// LS Electric XG5000 project: LoadWizardPro
// PLC LoadWizardPLC
// module base 0 slot 0: Input Module:XGI-D22A/B (DC 24V Input, 16 Contacts)
// module base 0 slot 1: Output Module:XGQ-RY2A/B (Relay Output, 16 Contacts (2A, No Varistor/Varistor))
// module base 0 slot 2: FEnet:XGL-EFMT(B) (Fast Ethernet Module, Electrical Master)
// module base 0 slot 0: Input/Output Module:XBE-DR16A (DC 24V Input, Relay Output, 16 Contacts)
// module base 0 slot 1: Input/Output Module:XBE-DR16A (DC 24V Input, Relay Output, 16 Contacts)

PROGRAM Main (task: Scan Program)

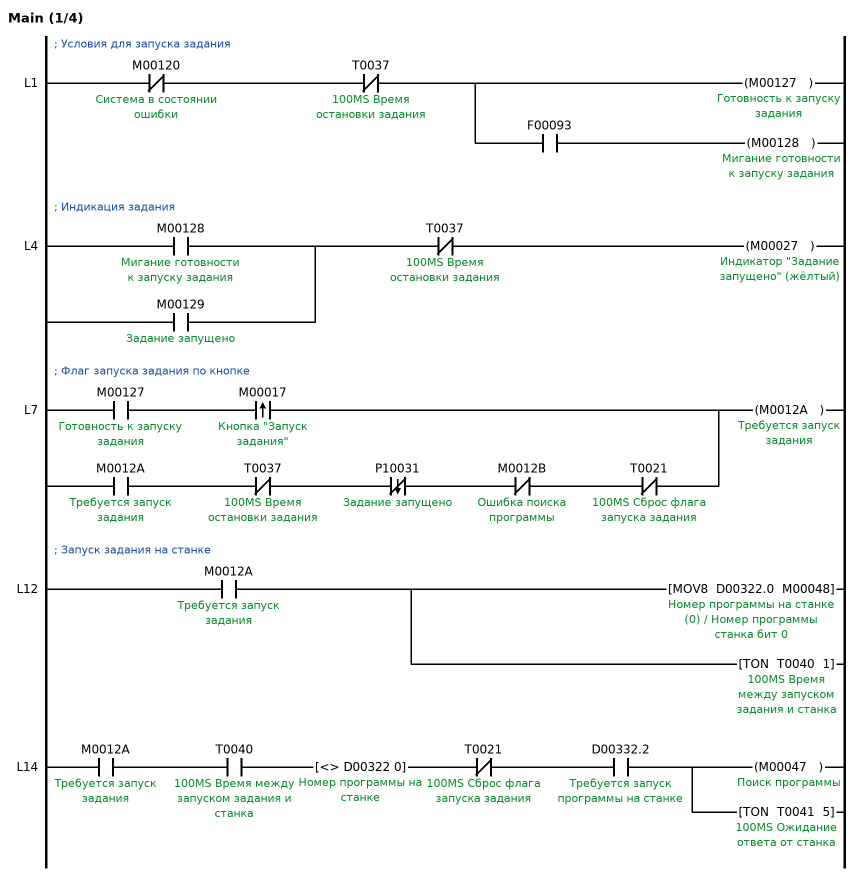
// Условия для запуска задания
; L1
LOAD NOT  M00120	// Система в состоянии ошибки
AND NOT   T0037	// 100MS Время остановки задания
OUT       M00127	// Готовность к запуску задания
AND       F00093
OUT       M00128	// Мигание готовности к запуску задания
// Индикация задания
; L4
LOAD      M00128	// Мигание готовности к запуску задания
OR        M00129	// Задание запущено
AND NOT   T0037	// 100MS Время остановки задания
OUT       M00027	// Индикатор "Задание запущено" (жёлтый)
// Флаг запуска задания по кнопке
; L7
LOAD      M00127	// Готовность к запуску задания
ANDP      M00017	// Кнопка "Запуск задания"
LOAD      M0012A	// Требуется запуск задания
AND NOT   T0037	// 100MS Время остановки задания
ANDN NOT  P10031	// Задание запущено
AND NOT   M0012B	// Ошибка поиска программы
AND NOT   T0021	// 100MS Сброс флага запуска задания
OR LOAD
OUT       M0012A	// Требуется запуск задания
// Запуск задания на станке
; L12
LOAD      M0012A	// Требуется запуск задания
MOV8      D00322.0 M00048	// Номер программы на станке (0) / Номер программы станка бит 0
TON       T0040 1	// 100MS Время между запуском задания и станка
; L14
LOAD      M0012A	// Требуется запуск задания
AND       T0040	// 100MS Время между запуском задания и станка
AND<>     D00322 0	// Номер программы на станке
AND NOT   T0021	// 100MS Сброс флага запуска задания
AND       D00332.2	// Требуется запуск программы на станке
OUT       M00047	// Поиск программы
TON       T0041 5	// 100MS Ожидание ответа от станка

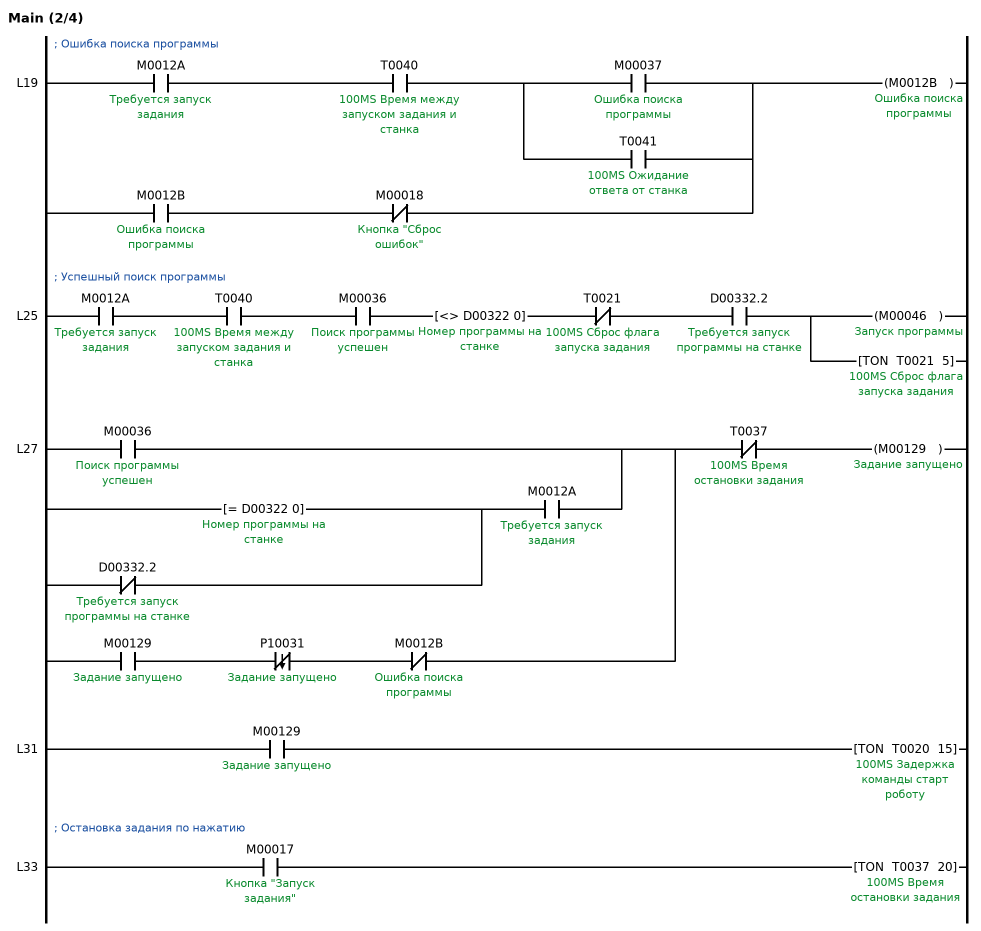
// Ошибка поиска программы
; L19
LOAD      M0012A	// Требуется запуск задания
AND       T0040	// 100MS Время между запуском задания и станка
LOAD      M00037	// Ошибка поиска программы
OR        T0041	// 100MS Ожидание ответа от станка
AND LOAD
LOAD      M0012B	// Ошибка поиска программы
AND NOT   M00018	// Кнопка "Сброс ошибок"
OR LOAD
OUT       M0012B	// Ошибка поиска программы
// Успешный поиск программы
; L25
LOAD      M0012A	// Требуется запуск задания
AND       T0040	// 100MS Время между запуском задания и станка
AND       M00036	// Поиск программы успешен
AND<>     D00322 0	// Номер программы на станке
AND NOT   T0021	// 100MS Сброс флага запуска задания
AND       D00332.2	// Требуется запуск программы на станке
OUT       M00046	// Запуск программы
TON       T0021 5	// 100MS Сброс флага запуска задания
; L27
LOAD      M00036	// Поиск программы успешен
LOAD=     D00322 0	// Номер программы на станке
OR NOT    D00332.2	// Требуется запуск программы на станке
AND       M0012A	// Требуется запуск задания
OR LOAD
LOAD      M00129	// Задание запущено
ANDN NOT  P10031	// Задание запущено
AND NOT   M0012B	// Ошибка поиска программы
OR LOAD
AND NOT   T0037	// 100MS Время остановки задания
OUT       M00129	// Задание запущено
; L31
LOAD      M00129	// Задание запущено
TON       T0020 15	// 100MS Задержка команды старт роботу
// Остановка задания по нажатию
; L33
LOAD      M00017	// Кнопка "Запуск задания"
TON       T0037 20	// 100MS Время остановки задания

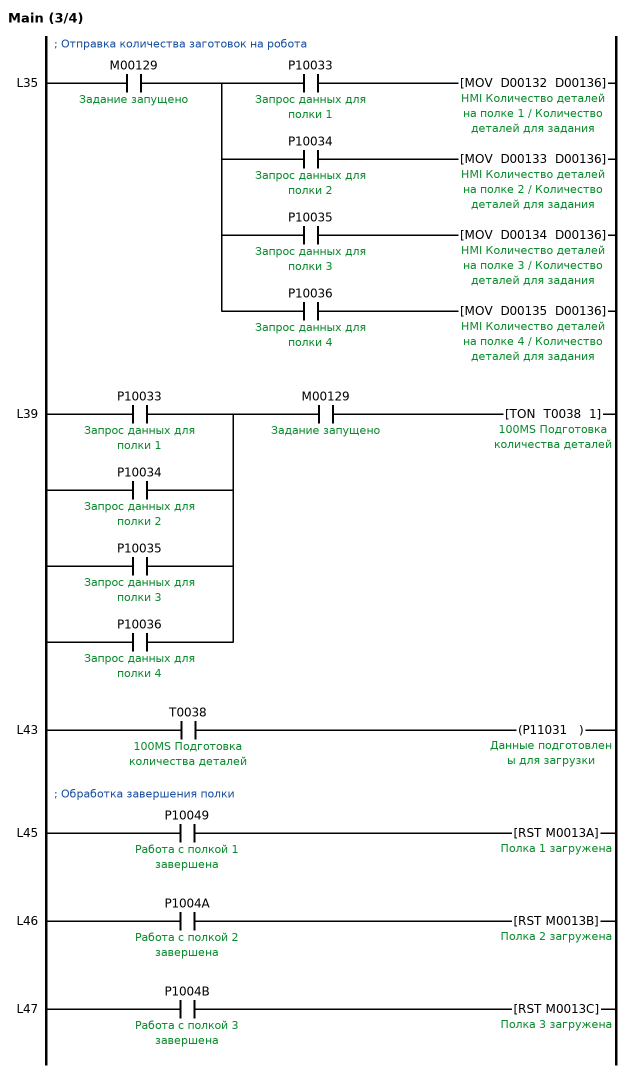
// Отправка количества заготовок на робота
; L35
LOAD      M00129	// Задание запущено
MPUSH
AND       P10033	// Запрос данных для полки 1
MOV       D00132 D00136	// HMI Количество деталей на полке 1 / Количество деталей для задания
MLOAD
AND       P10034	// Запрос данных для полки 2
MOV       D00133 D00136	// HMI Количество деталей на полке 2 / Количество деталей для задания
MLOAD
AND       P10035	// Запрос данных для полки 3
MOV       D00134 D00136	// HMI Количество деталей на полке 3 / Количество деталей для задания
MPOP
AND       P10036	// Запрос данных для полки 4
MOV       D00135 D00136	// HMI Количество деталей на полке 4 / Количество деталей для задания
; L39
LOAD      P10033	// Запрос данных для полки 1
OR        P10034	// Запрос данных для полки 2
OR        P10035	// Запрос данных для полки 3
OR        P10036	// Запрос данных для полки 4
AND       M00129	// Задание запущено
TON       T0038 1	// 100MS Подготовка количества деталей
; L43
LOAD      T0038	// 100MS Подготовка количества деталей
OUT       P11031	// Данные подготовлены для загрузки
// Обработка завершения полки
; L45
LOAD      P10049	// Работа с полкой 1 завершена
RST       M0013A	// Полка 1 загружена
; L46
LOAD      P1004A	// Работа с полкой 2 завершена
RST       M0013B	// Полка 2 загружена
; L47
LOAD      P1004B	// Работа с полкой 3 завершена
RST       M0013C	// Полка 3 загружена

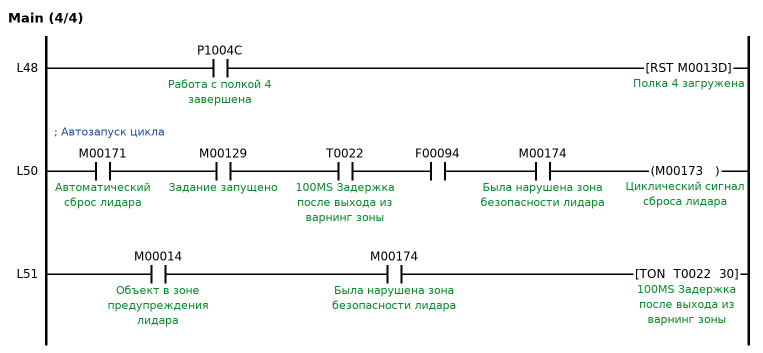
; L48
LOAD      P1004C	// Работа с полкой 4 завершена
RST       M0013D	// Полка 4 загружена
// Автозапуск цикла
; L50
LOAD      M00171	// Автоматический сброс лидара
AND       M00129	// Задание запущено
AND       T0022	// 100MS Задержка после выхода из варнинг зоны
AND       F00094
AND       M00174	// Была нарушена зона безопасности лидара
OUT       M00173	// Циклический сигнал сброса лидара
; L51
LOAD      M00014	// Объект в зоне предупреждения лидара
AND       M00174	// Была нарушена зона безопасности лидара
TON       T0022 30	// 100MS Задержка после выхода из варнинг зоны

PROGRAM Robot (task: Scan Program)

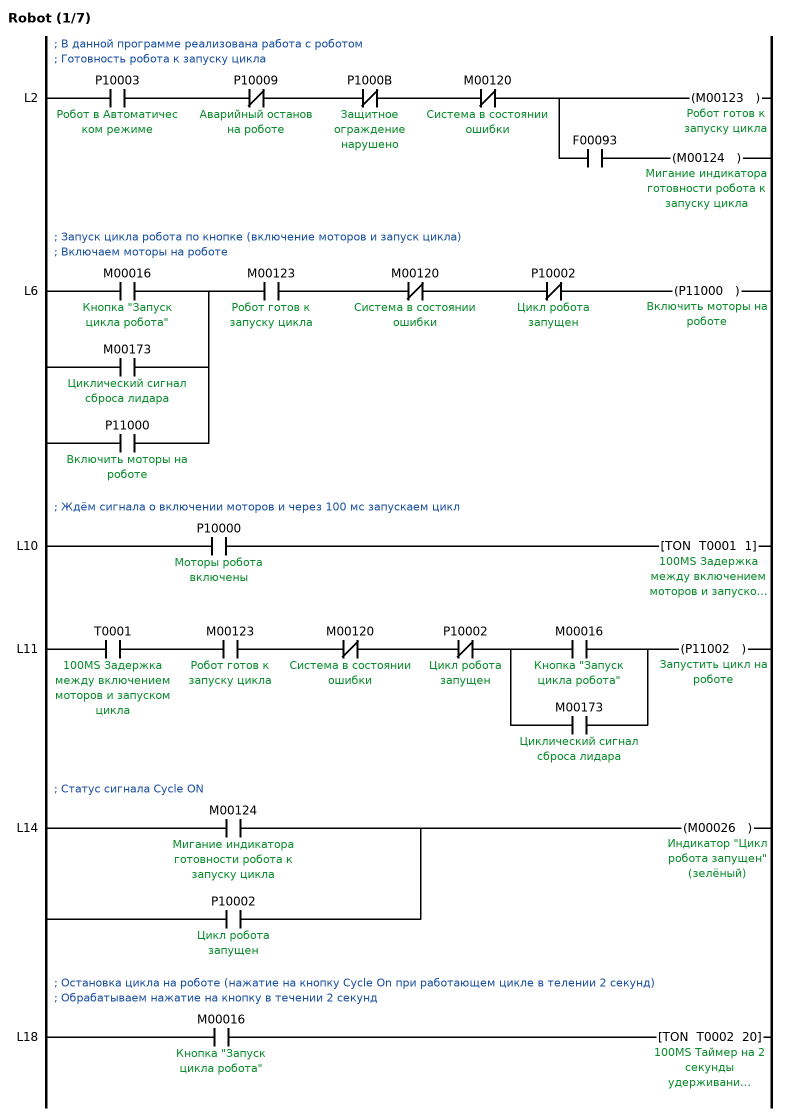
// В данной программе реализована работа с роботом
// Готовность робота к запуску цикла
; L2
LOAD      P10003	// Робот в Автоматическом режиме
AND NOT   P10009	// Аварийный останов на роботе
AND NOT   P1000B	// Защитное ограждение нарушено
AND NOT   M00120	// Система в состоянии ошибки
OUT       M00123	// Робот готов к запуску цикла
AND       F00093
OUT       M00124	// Мигание индикатора готовности робота к запуску цикла
// Запуск цикла робота по кнопке (включение моторов и запуск цикла)
// Включаем моторы на роботе
; L6
LOAD      M00016	// Кнопка "Запуск цикла робота"
OR        M00173	// Циклический сигнал сброса лидара
OR        P11000	// Включить моторы на роботе
AND       M00123	// Робот готов к запуску цикла
AND NOT   M00120	// Система в состоянии ошибки
AND NOT   P10002	// Цикл робота запущен
OUT       P11000	// Включить моторы на роботе
// Ждём сигнала о включении моторов и через 100 мс запускаем цикл
; L10
LOAD      P10000	// Моторы робота включены
TON       T0001 1	// 100MS Задержка между включением моторов и запуском цикла
; L11
LOAD      T0001	// 100MS Задержка между включением моторов и запуском цикла
AND       M00123	// Робот готов к запуску цикла
AND NOT   M00120	// Система в состоянии ошибки
AND NOT   P10002	// Цикл робота запущен
LOAD      M00016	// Кнопка "Запуск цикла робота"
OR        M00173	// Циклический сигнал сброса лидара
AND LOAD
OUT       P11002	// Запустить цикл на роботе
// output comment: 
// Статус сигнала Cycle ON
; L14
LOAD      M00124	// Мигание индикатора готовности робота к запуску цикла
OR        P10002	// Цикл робота запущен
OUT       M00026	// Индикатор "Цикл робота запущен" (зелёный)
// Остановка цикла на роботе (нажатие на кнопку Cycle On при работающем цикле в телении 2 секунд)
// Обрабатываем нажатие на кнопку в течении 2 секунд
; L18
LOAD      M00016	// Кнопка "Запуск цикла робота"
TON       T0002 20	// 100MS Таймер на 2 секунды удерживания кнопки

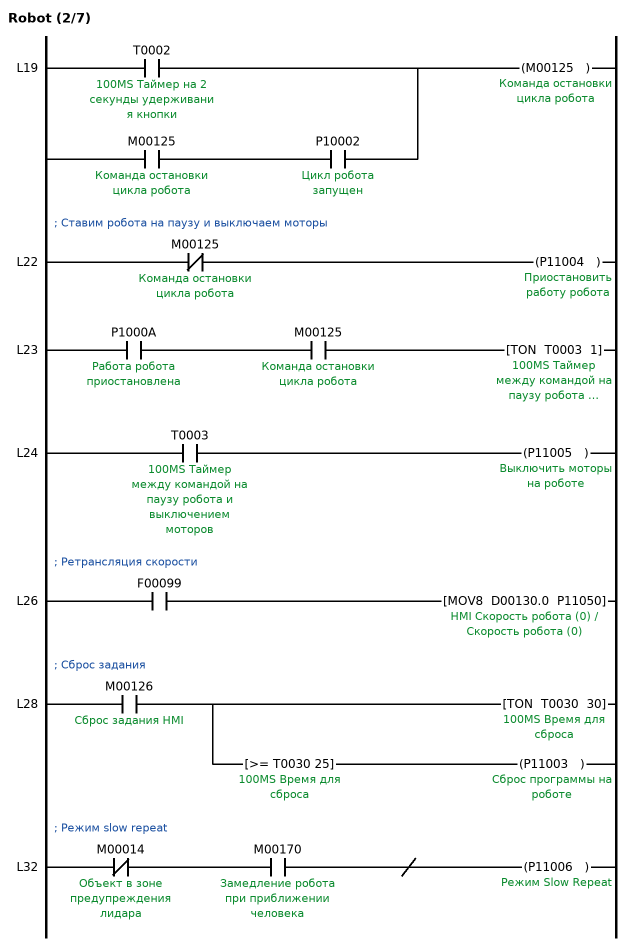
; L19
LOAD      T0002	// 100MS Таймер на 2 секунды удерживания кнопки
LOAD      M00125	// Команда остановки цикла робота
AND       P10002	// Цикл робота запущен
OR LOAD
OUT       M00125	// Команда остановки цикла робота
// Ставим робота на паузу и выключаем моторы
; L22
LOAD NOT  M00125	// Команда остановки цикла робота
OUT       P11004	// Приостановить работу робота
; L23
LOAD      P1000A	// Работа робота приостановлена
AND       M00125	// Команда остановки цикла робота
TON       T0003 1	// 100MS Таймер между командой на паузу робота и выключением моторов
; L24
LOAD      T0003	// 100MS Таймер между командой на паузу робота и выключением моторов
OUT       P11005	// Выключить моторы на роботе
// Ретрансляция скорости
; L26
LOAD      F00099
MOV8      D00130.0 P11050	// HMI Скорость робота (0) / Скорость робота (0)
// Сброс задания
; L28
LOAD      M00126	// Сброс задания HMI
TON       T0030 30	// 100MS Время для сброса
AND>=     T0030 25	// 100MS Время для сброса
OUT       P11003	// Сброс программы на роботе
// Режим slow repeat
; L32
LOAD NOT  M00014	// Объект в зоне предупреждения лидара
AND       M00170	// Замедление робота при приближении человека
NOT
OUT       P11006	// Режим Slow Repeat

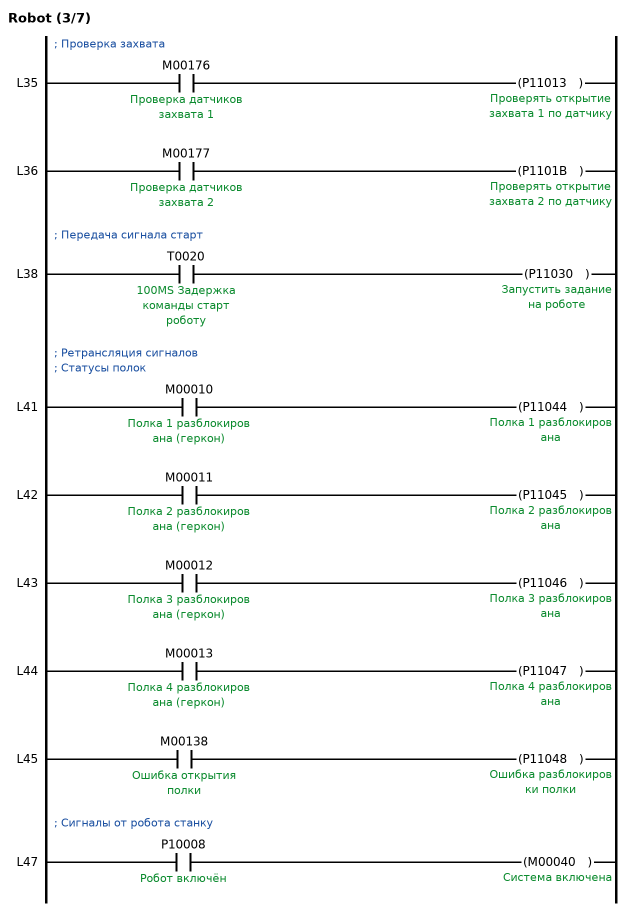
// Проверка захвата
; L35
LOAD      M00176	// Проверка датчиков захвата 1
OUT       P11013	// Проверять открытие захвата 1 по датчику
; L36
LOAD      M00177	// Проверка датчиков захвата 2
OUT       P1101B	// Проверять открытие захвата 2 по датчику
// Передача сигнала старт
; L38
LOAD      T0020	// 100MS Задержка команды старт роботу
OUT       P11030	// Запустить задание на роботе
// Ретрансляция сигналов
// Статусы полок
; L41
LOAD      M00010	// Полка 1 разблокирована (геркон)
OUT       P11044	// Полка 1 разблокирована
; L42
LOAD      M00011	// Полка 2 разблокирована (геркон)
OUT       P11045	// Полка 2 разблокирована
; L43
LOAD      M00012	// Полка 3 разблокирована (геркон)
OUT       P11046	// Полка 3 разблокирована
; L44
LOAD      M00013	// Полка 4 разблокирована (геркон)
OUT       P11047	// Полка 4 разблокирована
; L45
LOAD      M00138	// Ошибка открытия полки
OUT       P11048	// Ошибка разблокировки полки
// Сигналы от робота станку
; L47
LOAD      P10008	// Робот включён
OUT       M00040	// Система включена

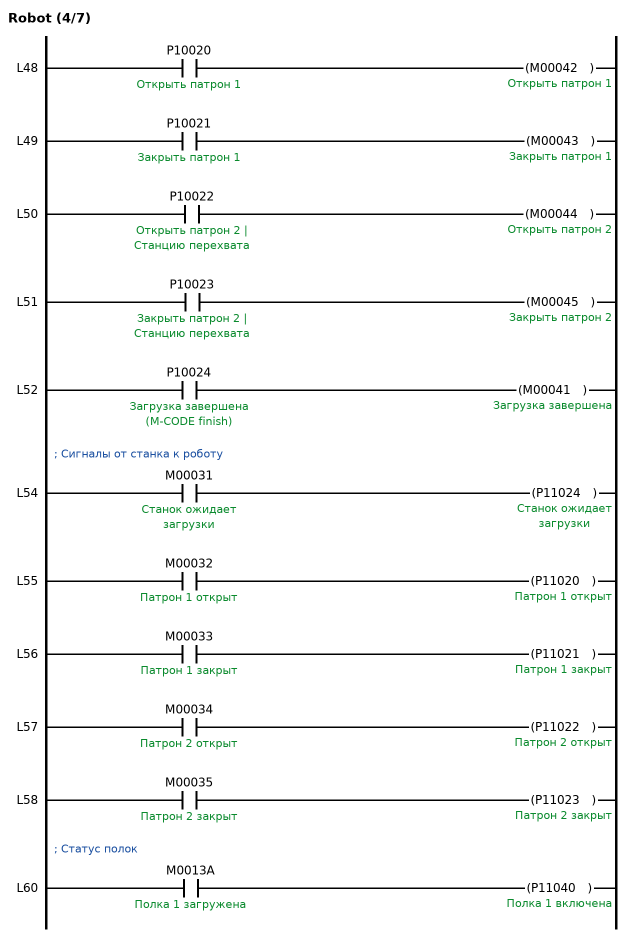
; L48
LOAD      P10020	// Открыть патрон 1
OUT       M00042	// Открыть патрон 1
; L49
LOAD      P10021	// Закрыть патрон 1
OUT       M00043	// Закрыть патрон 1
; L50
LOAD      P10022	// Открыть патрон 2 | Cтанцию перехвата
OUT       M00044	// Открыть патрон 2
; L51
LOAD      P10023	// Закрыть патрон 2 | Cтанцию перехвата
OUT       M00045	// Закрыть патрон 2
; L52
LOAD      P10024	// Загрузка завершена (M-CODE finish)
OUT       M00041	// Загрузка завершена
// Сигналы от станка к роботу
; L54
LOAD      M00031	// Станок ожидает загрузки
OUT       P11024	// Станок ожидает загрузки
; L55
LOAD      M00032	// Патрон 1 открыт
OUT       P11020	// Патрон 1 открыт
; L56
LOAD      M00033	// Патрон 1 закрыт
OUT       P11021	// Патрон 1 закрыт
; L57
LOAD      M00034	// Патрон 2 открыт
OUT       P11022	// Патрон 2 открыт
; L58
LOAD      M00035	// Патрон 2 закрыт
OUT       P11023	// Патрон 2 закрыт
// Статус полок
; L60
LOAD      M0013A	// Полка 1 загружена
OUT       P11040	// Полка 1 включена

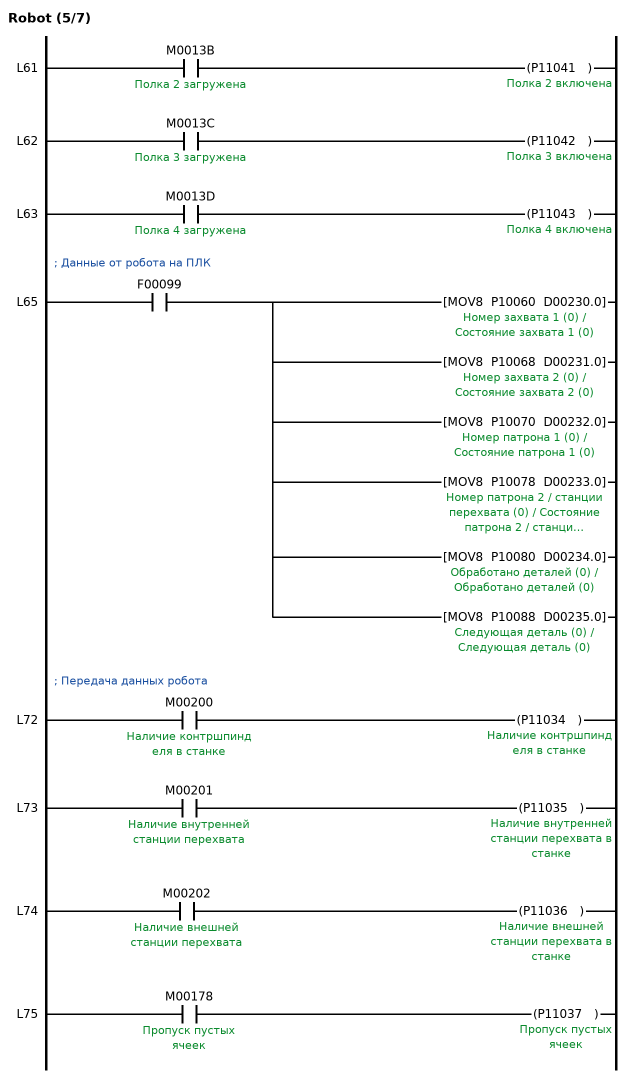
; L61
LOAD      M0013B	// Полка 2 загружена
OUT       P11041	// Полка 2 включена
; L62
LOAD      M0013C	// Полка 3 загружена
OUT       P11042	// Полка 3 включена
; L63
LOAD      M0013D	// Полка 4 загружена
OUT       P11043	// Полка 4 включена
// Данные от робота на ПЛК
; L65
LOAD      F00099
MOV8      P10060 D00230.0	// Номер захвата 1 (0) / Состояние захвата 1 (0)
MOV8      P10068 D00231.0	// Номер захвата 2 (0) / Состояние захвата 2 (0)
MOV8      P10070 D00232.0	// Номер патрона 1 (0) / Состояние патрона 1 (0)
MOV8      P10078 D00233.0	// Номер патрона 2 / станции перехвата (0) / Состояние патрона 2 / станции перехвата (0)
MOV8      P10080 D00234.0	// Обработано деталей (0) / Обработано деталей (0)
MOV8      P10088 D00235.0	// Следующая деталь (0) / Следующая деталь (0)
// Передача данных робота
; L72
LOAD      M00200	// Наличие контршпинделя в станке
OUT       P11034	// Наличие контршпинделя в станке
; L73
LOAD      M00201	// Наличие внутренней станции перехвата
OUT       P11035	// Наличие внутренней станции перехвата в станке
; L74
LOAD      M00202	// Наличие внешней станции перехвата
OUT       P11036	// Наличие внешней станции перехвата в станке
; L75
LOAD      M00178	// Пропуск пустых ячеек
OUT       P11037	// Пропуск пустых ячеек

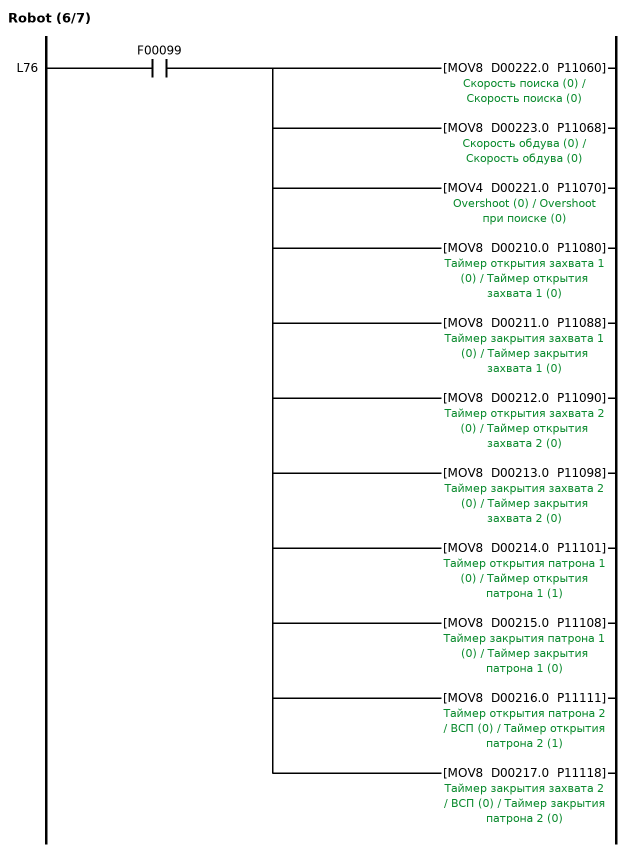
; L76
LOAD      F00099
MOV8      D00222.0 P11060	// Скорость поиска (0) / Скорость поиска (0)
MOV8      D00223.0 P11068	// Скорость обдува (0) / Скорость обдува (0)
MOV4      D00221.0 P11070	// Overshoot (0) / Overshoot при поиске (0)
MOV8      D00210.0 P11080	// Таймер открытия захвата 1 (0) / Таймер открытия захвата 1 (0)
MOV8      D00211.0 P11088	// Таймер закрытия захвата 1 (0) / Таймер закрытия захвата 1 (0)
MOV8      D00212.0 P11090	// Таймер открытия захвата 2 (0) / Таймер открытия захвата 2 (0)
MOV8      D00213.0 P11098	// Таймер закрытия захвата 2 (0) / Таймер закрытия захвата 2 (0)
MOV8      D00214.0 P11101	// Таймер открытия патрона 1 (0) / Таймер открытия патрона 1 (1)
MOV8      D00215.0 P11108	// Таймер закрытия патрона 1 (0) / Таймер закрытия патрона 1 (0)
MOV8      D00216.0 P11111	// Таймер открытия патрона 2 / ВСП (0) / Таймер открытия патрона 2 (1)
MOV8      D00217.0 P11118	// Таймер закрытия захвата 2 / ВСП (0) / Таймер закрытия патрона 2 (0)

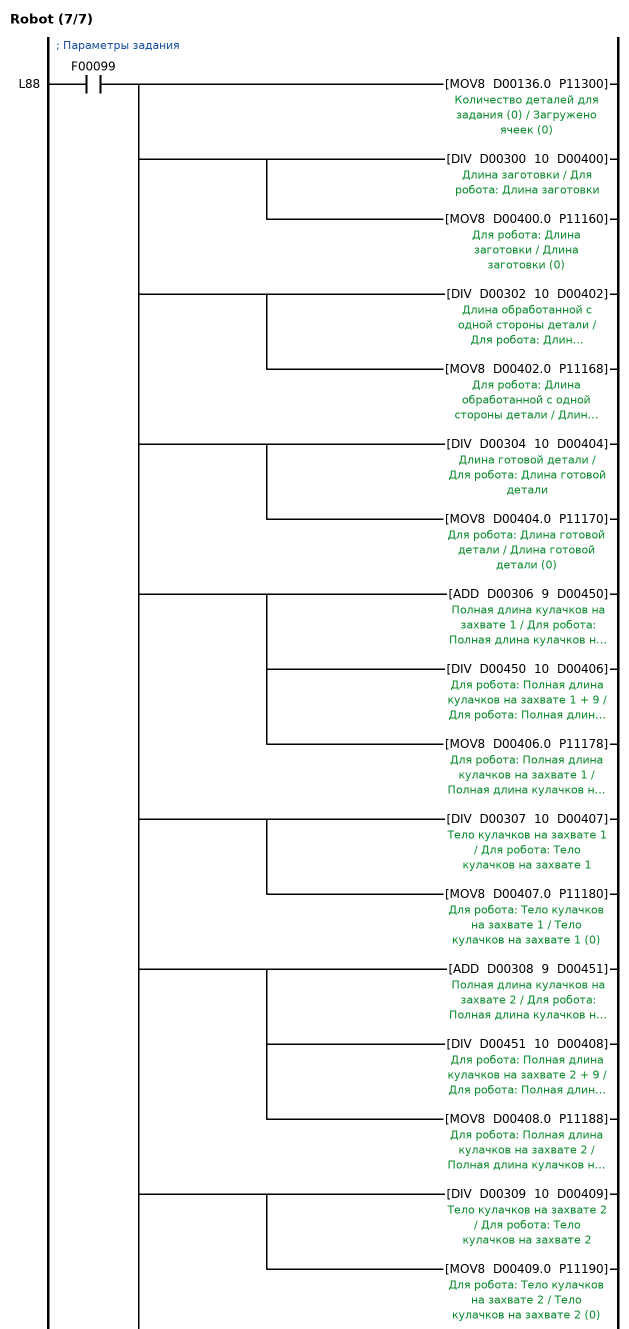

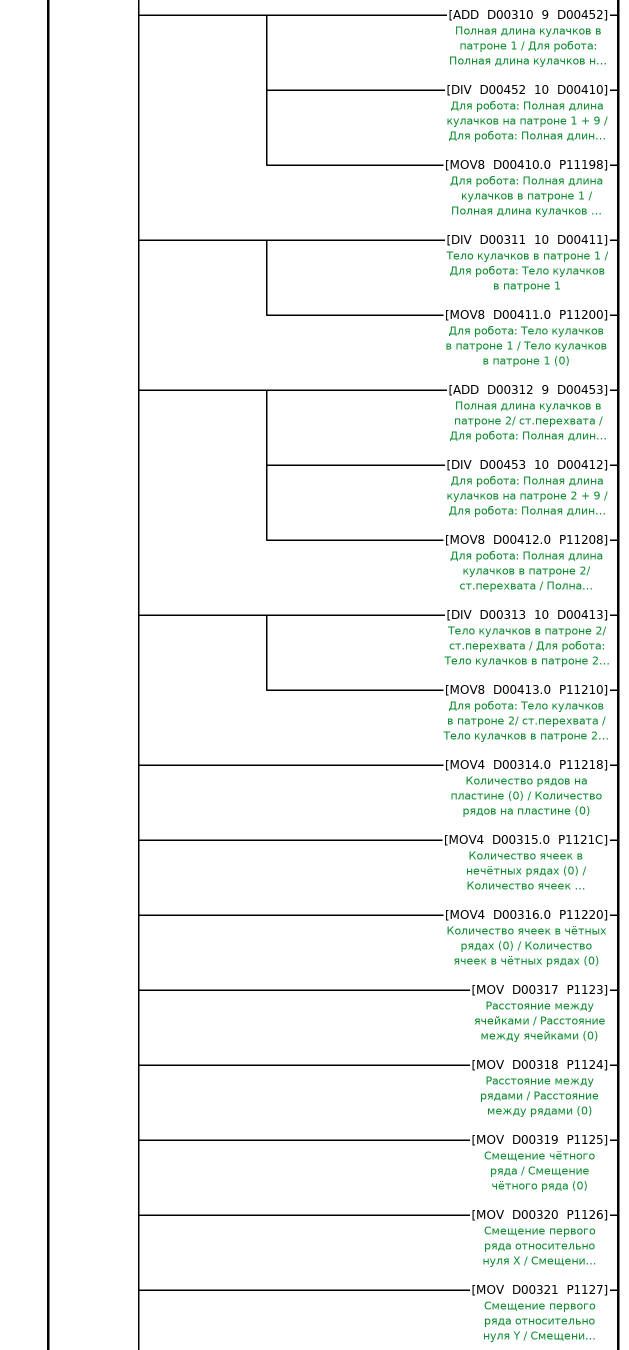

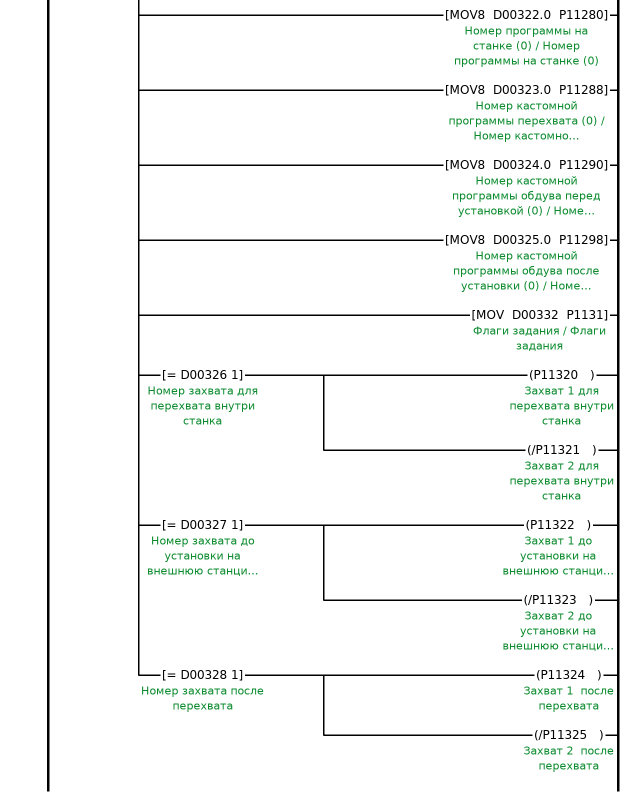
// Параметры задания
; L88
LOAD      F00099
MOV8      D00136.0 P11300	// Количество деталей для задания (0) / Загружено ячеек (0)
DIV       D00300 10 D00400	// Длина заготовки / Для робота: Длина заготовки
MOV8      D00400.0 P11160	// Для робота: Длина заготовки / Длина заготовки (0)
DIV       D00302 10 D00402	// Длина обработанной с одной стороны детали / Для робота: Длина обработанной с одной стороны детали
MOV8      D00402.0 P11168	// Для робота: Длина обработанной с одной стороны детали / Длина обработанной с одной стороны детали (0)
DIV       D00304 10 D00404	// Длина готовой детали / Для робота: Длина готовой детали
MOV8      D00404.0 P11170	// Для робота: Длина готовой детали / Длина готовой детали (0)
ADD       D00306 9 D00450	// Полная длина кулачков на захвате 1 / Для робота: Полная длина кулачков на захвате 1 + 9
DIV       D00450 10 D00406	// Для робота: Полная длина кулачков на захвате 1 + 9 / Для робота: Полная длина кулачков на захвате 1
MOV8      D00406.0 P11178	// Для робота: Полная длина кулачков на захвате 1 / Полная длина кулачков на захвате 1 (0)
DIV       D00307 10 D00407	// Тело кулачков на захвате 1 / Для робота: Тело кулачков на захвате 1
MOV8      D00407.0 P11180	// Для робота: Тело кулачков на захвате 1 / Тело кулачков на захвате 1 (0)
ADD       D00308 9 D00451	// Полная длина кулачков на захвате 2 / Для робота: Полная длина кулачков на захвате 2 + 9
DIV       D00451 10 D00408	// Для робота: Полная длина кулачков на захвате 2 + 9 / Для робота: Полная длина кулачков на захвате 2
MOV8      D00408.0 P11188	// Для робота: Полная длина кулачков на захвате 2 / Полная длина кулачков на захвате 2 (0)
DIV       D00309 10 D00409	// Тело кулачков на захвате 2 / Для робота: Тело кулачков на захвате 2
MOV8      D00409.0 P11190	// Для робота: Тело кулачков на захвате 2 / Тело кулачков на захвате 2 (0)
ADD       D00310 9 D00452	// Полная длина кулачков в патроне 1 / Для робота: Полная длина кулачков на патроне 1 + 9
DIV       D00452 10 D00410	// Для робота: Полная длина кулачков на патроне 1 + 9 / Для робота: Полная длина кулачков в патроне 1
MOV8      D00410.0 P11198	// Для робота: Полная длина кулачков в патроне 1 / Полная длина кулачков в патроне 1 (0)
DIV       D00311 10 D00411	// Тело кулачков в патроне 1 / Для робота: Тело кулачков в патроне 1
MOV8      D00411.0 P11200	// Для робота: Тело кулачков в патроне 1 / Тело кулачков в патроне 1 (0)
ADD       D00312 9 D00453	// Полная длина кулачков в патроне 2/ ст.перехвата / Для робота: Полная длина кулачков на патроне 2 + 9
DIV       D00453 10 D00412	// Для робота: Полная длина кулачков на патроне 2 + 9 / Для робота: Полная длина кулачков в патроне 2/ ст.перехвата
MOV8      D00412.0 P11208	// Для робота: Полная длина кулачков в патроне 2/ ст.перехвата / Полная длина кулачков в патроне 2/ ст.перехвата (0)
DIV       D00313 10 D00413	// Тело кулачков в патроне 2/ ст.перехвата / Для робота: Тело кулачков в патроне 2/ ст.перехвата
MOV8      D00413.0 P11210	// Для робота: Тело кулачков в патроне 2/ ст.перехвата / Тело кулачков в патроне 2/ ст.перехвата  (0)
MOV4      D00314.0 P11218	// Количество рядов на пластине (0) / Количество рядов на пластине (0)
MOV4      D00315.0 P1121C	// Количество ячеек в нечётных рядах (0) / Количество ячеек в нечётных рядах (0)
MOV4      D00316.0 P11220	// Количество ячеек в чётных рядах (0) / Количество ячеек в чётных рядах (0)
MOV       D00317 P1123	// Расстояние между ячейками / Расстояние между ячейками (0)
MOV       D00318 P1124	// Расстояние между рядами / Расстояние между рядами (0)
MOV       D00319 P1125	// Смещение чётного ряда / Смещение чётного ряда (0)
MOV       D00320 P1126	// Смещение первого ряда относительно нуля Х / Смещение первого ряда относительно нуля Х (0)
MOV       D00321 P1127	// Смещение первого ряда относительно нуля Y / Смещение первого ряда относительно нуля Y (0)
MOV8      D00322.0 P11280	// Номер программы на станке (0) / Номер программы на станке (0)
MOV8      D00323.0 P11288	// Номер кастомной программы перехвата (0) / Номер кастомной программы перехвата 1 (0)
MOV8      D00324.0 P11290	// Номер кастомной программы обдува перед установкой (0) / Номер программы обдува 1 (0)
MOV8      D00325.0 P11298	// Номер кастомной программы обдува после установки (0) / Номер программы обдува 2 (0)
MOV       D00332 P1131	// Флаги задания / Флаги задания
MPUSH
AND=      D00326 1	// Номер захвата для перехвата внутри станка
OUT       P11320	// Захват 1 для перехвата внутри станка 
OUT NOT   P11321	// Захват 2 для перехвата внутри станка 
MLOAD
AND=      D00327 1	// Номер захвата до установки на внешнюю станцию перехвата
OUT       P11322	// Захват 1 до установки на внешнюю станцию перехвата
OUT NOT   P11323	// Захват 2 до установки на внешнюю станцию перехвата
MPOP
AND=      D00328 1	// Номер захвата после перехвата
OUT       P11324	// Захват 1  после перехвата
OUT NOT   P11325	// Захват 2  после перехвата

PROGRAM IO (task: Scan Program)

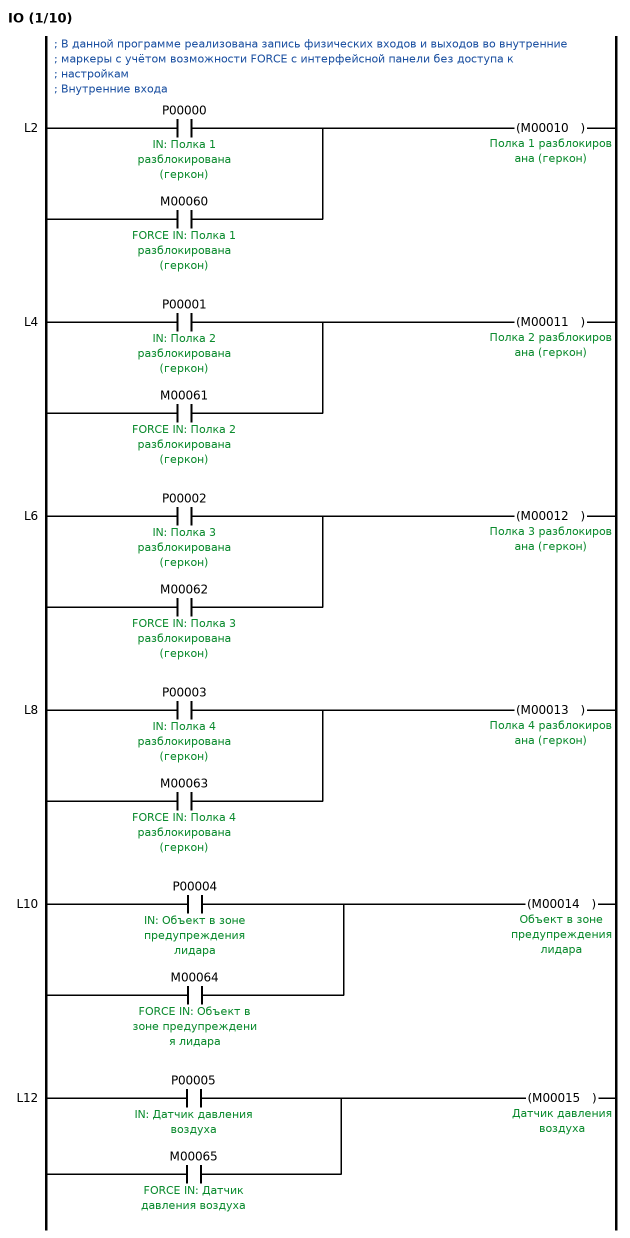
// В данной программе реализована запись физических входов и выходов во внутренние маркеры с учётом возможности FORCE с интерфейсной панели без доступа к настройкам
// Внутренние входа
; L2
LOAD      P00000	// IN: Полка 1 разблокирована (геркон)
OR        M00060	// FORCE IN: Полка 1 разблокирована (геркон)
OUT       M00010	// Полка 1 разблокирована (геркон)
; L4
LOAD      P00001	// IN: Полка 2 разблокирована (геркон)
OR        M00061	// FORCE IN: Полка 2 разблокирована (геркон)
OUT       M00011	// Полка 2 разблокирована (геркон)
; L6
LOAD      P00002	// IN: Полка 3 разблокирована (геркон)
OR        M00062	// FORCE IN: Полка 3 разблокирована (геркон)
OUT       M00012	// Полка 3 разблокирована (геркон)
; L8
LOAD      P00003	// IN: Полка 4 разблокирована (геркон)
OR        M00063	// FORCE IN: Полка 4 разблокирована (геркон)
OUT       M00013	// Полка 4 разблокирована (геркон)
; L10
LOAD      P00004	// IN: Объект в зоне предупреждения лидара
OR        M00064	// FORCE IN: Объект в зоне предупреждения лидара
OUT       M00014	// Объект в зоне предупреждения лидара
; L12
LOAD      P00005	// IN: Датчик давления воздуха
OR        M00065	// FORCE IN: Датчик давления воздуха
OUT       M00015	// Датчик давления воздуха

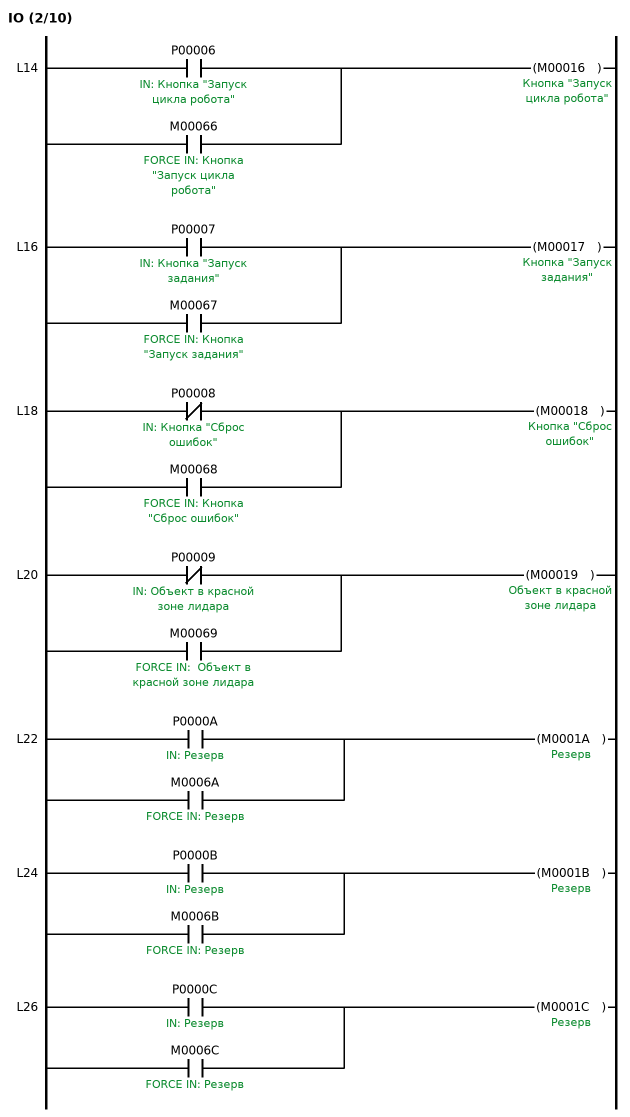
; L14
LOAD      P00006	// IN: Кнопка "Запуск цикла робота"
OR        M00066	// FORCE IN: Кнопка "Запуск цикла робота"
OUT       M00016	// Кнопка "Запуск цикла робота"
; L16
LOAD      P00007	// IN: Кнопка "Запуск задания"
OR        M00067	// FORCE IN: Кнопка "Запуск задания"
OUT       M00017	// Кнопка "Запуск задания"
; L18
LOAD NOT  P00008	// IN: Кнопка "Сброс ошибок"
OR        M00068	// FORCE IN: Кнопка "Сброс ошибок"
OUT       M00018	// Кнопка "Сброс ошибок"
; L20
LOAD NOT  P00009	// IN: Объект в красной зоне лидара
OR        M00069	// FORCE IN:  Объект в красной зоне лидара
OUT       M00019	//  Объект в красной зоне лидара
; L22
LOAD      P0000A	// IN: Резерв
OR        M0006A	// FORCE IN: Резерв
OUT       M0001A	// Резерв
; L24
LOAD      P0000B	// IN: Резерв
OR        M0006B	// FORCE IN: Резерв
OUT       M0001B	// Резерв
; L26
LOAD      P0000C	// IN: Резерв
OR        M0006C	// FORCE IN: Резерв
OUT       M0001C	// Резерв

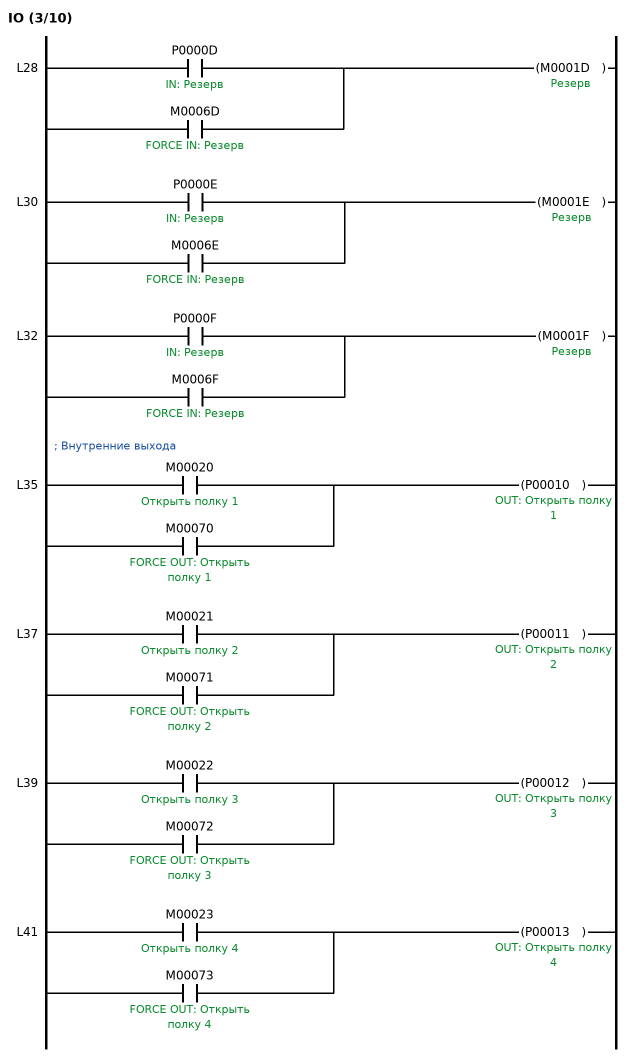
; L28
LOAD      P0000D	// IN: Резерв
OR        M0006D	// FORCE IN: Резерв
OUT       M0001D	// Резерв
; L30
LOAD      P0000E	// IN: Резерв
OR        M0006E	// FORCE IN: Резерв
OUT       M0001E	// Резерв
; L32
LOAD      P0000F	// IN: Резерв
OR        M0006F	// FORCE IN: Резерв
OUT       M0001F	// Резерв
// Внутренние выхода
; L35
LOAD      M00020	// Открыть полку 1
OR        M00070	// FORCE OUT: Открыть полку 1
OUT       P00010	// OUT: Открыть полку 1
; L37
LOAD      M00021	// Открыть полку 2
OR        M00071	// FORCE OUT: Открыть полку 2
OUT       P00011	// OUT: Открыть полку 2
; L39
LOAD      M00022	// Открыть полку 3
OR        M00072	// FORCE OUT: Открыть полку 3
OUT       P00012	// OUT: Открыть полку 3
; L41
LOAD      M00023	// Открыть полку 4
OR        M00073	// FORCE OUT: Открыть полку 4
OUT       P00013	// OUT: Открыть полку 4

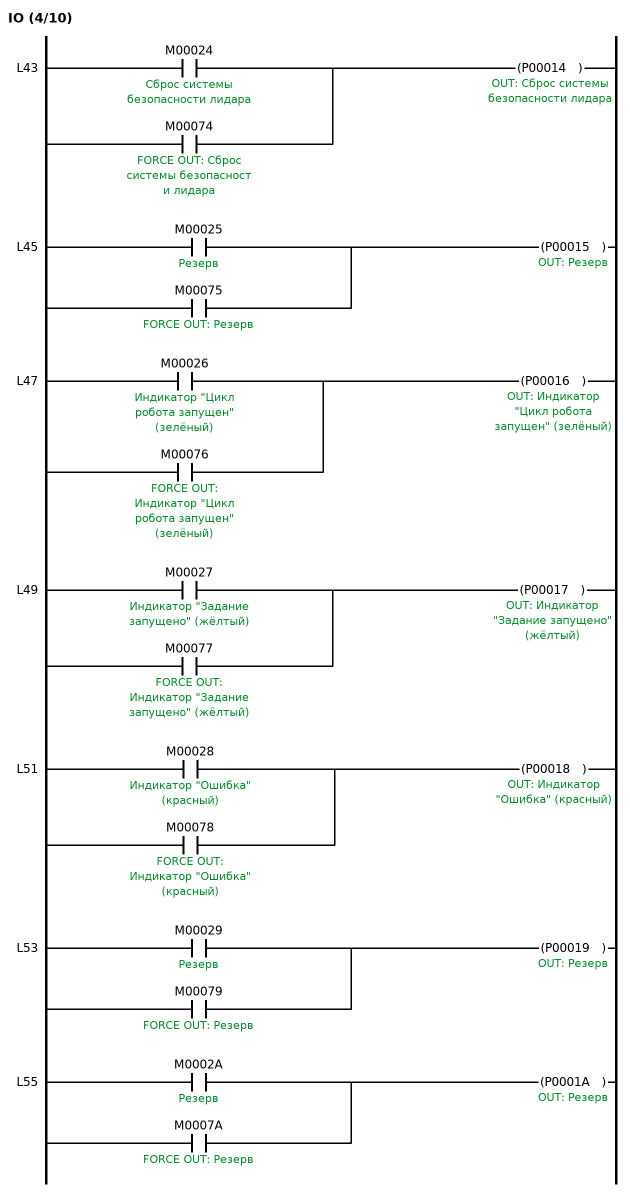
; L43
LOAD      M00024	// Сброс системы безопасности лидара
OR        M00074	// FORCE OUT: Сброс системы безопасности лидара
OUT       P00014	// OUT: Сброс системы безопасности лидара
; L45
LOAD      M00025	// Резерв
OR        M00075	// FORCE OUT: Резерв
OUT       P00015	// OUT: Резерв
; L47
LOAD      M00026	// Индикатор "Цикл робота запущен" (зелёный)
OR        M00076	// FORCE OUT: Индикатор "Цикл робота запущен" (зелёный)
OUT       P00016	// OUT: Индикатор "Цикл робота запущен" (зелёный)
; L49
LOAD      M00027	// Индикатор "Задание запущено" (жёлтый)
OR        M00077	// FORCE OUT: Индикатор "Задание запущено" (жёлтый)
OUT       P00017	// OUT: Индикатор "Задание запущено" (жёлтый)
; L51
LOAD      M00028	// Индикатор "Ошибка" (красный)
OR        M00078	// FORCE OUT: Индикатор "Ошибка" (красный)
OUT       P00018	// OUT: Индикатор "Ошибка" (красный)
; L53
LOAD      M00029	// Резерв
OR        M00079	// FORCE OUT: Резерв
OUT       P00019	// OUT: Резерв
; L55
LOAD      M0002A	// Резерв
OR        M0007A	// FORCE OUT: Резерв
OUT       P0001A	// OUT: Резерв

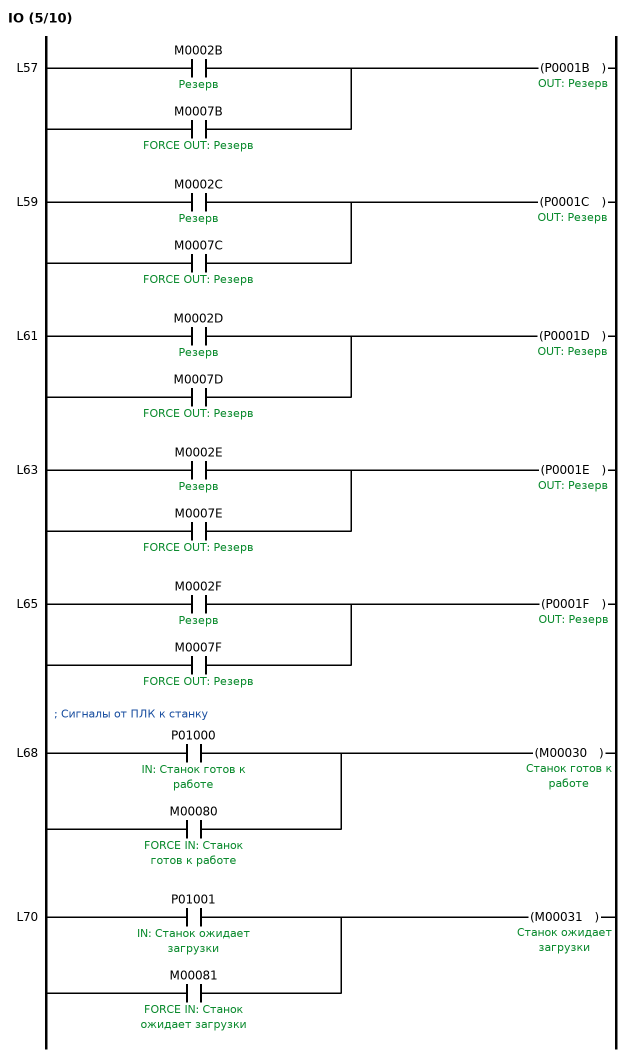
; L57
LOAD      M0002B	// Резерв
OR        M0007B	// FORCE OUT: Резерв
OUT       P0001B	// OUT: Резерв
; L59
LOAD      M0002C	// Резерв
OR        M0007C	// FORCE OUT: Резерв
OUT       P0001C	// OUT: Резерв
; L61
LOAD      M0002D	// Резерв
OR        M0007D	// FORCE OUT: Резерв
OUT       P0001D	// OUT: Резерв
; L63
LOAD      M0002E	// Резерв
OR        M0007E	// FORCE OUT: Резерв
OUT       P0001E	// OUT: Резерв
; L65
LOAD      M0002F	// Резерв
OR        M0007F	// FORCE OUT: Резерв
OUT       P0001F	// OUT: Резерв
// Сигналы от ПЛК к станку
; L68
LOAD      P01000	// IN: Станок готов к работе
OR        M00080	// FORCE IN: Станок готов к работе
OUT       M00030	// Станок готов к работе
; L70
LOAD      P01001	// IN: Станок ожидает загрузки
OR        M00081	// FORCE IN: Станок ожидает загрузки
OUT       M00031	// Станок ожидает загрузки

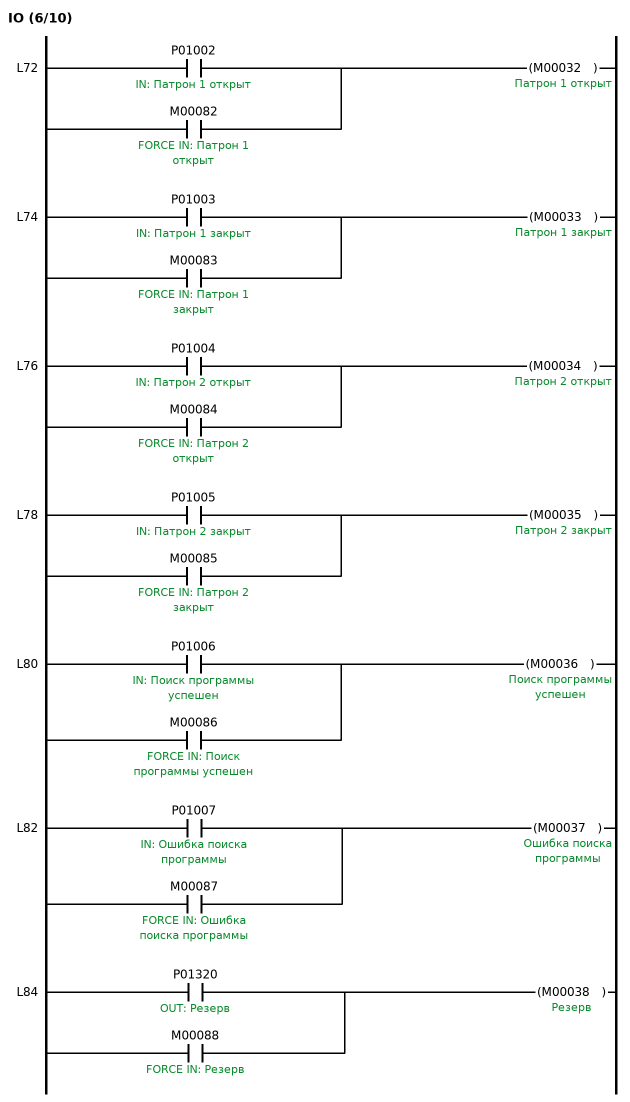
; L72
LOAD      P01002	// IN: Патрон 1 открыт
OR        M00082	// FORCE IN: Патрон 1 открыт
OUT       M00032	// Патрон 1 открыт
; L74
LOAD      P01003	// IN: Патрон 1 закрыт
OR        M00083	// FORCE IN: Патрон 1 закрыт
OUT       M00033	// Патрон 1 закрыт
; L76
LOAD      P01004	// IN: Патрон 2 открыт
OR        M00084	// FORCE IN: Патрон 2 открыт
OUT       M00034	// Патрон 2 открыт
; L78
LOAD      P01005	// IN: Патрон 2 закрыт
OR        M00085	// FORCE IN: Патрон 2 закрыт
OUT       M00035	// Патрон 2 закрыт
; L80
LOAD      P01006	// IN: Поиск программы успешен
OR        M00086	// FORCE IN: Поиск программы успешен
OUT       M00036	// Поиск программы успешен
; L82
LOAD      P01007	// IN: Ошибка поиска программы
OR        M00087	// FORCE IN: Ошибка поиска программы
OUT       M00037	// Ошибка поиска программы
; L84
LOAD      P01320	// OUT: Резерв
OR        M00088	// FORCE IN: Резерв
OUT       M00038	// Резерв

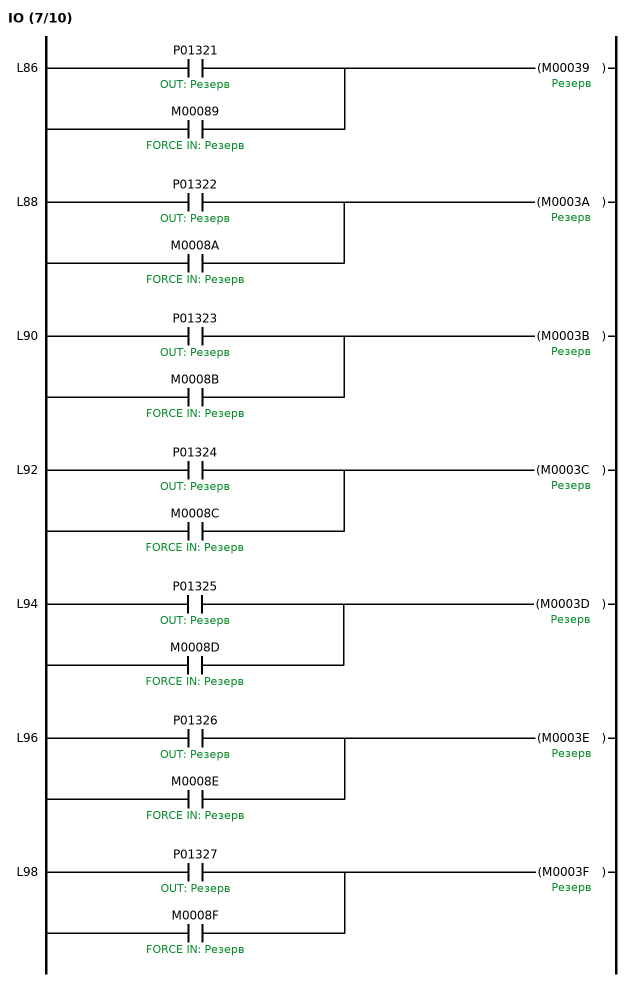
; L86
LOAD      P01321	// OUT: Резерв
OR        M00089	// FORCE IN: Резерв
OUT       M00039	// Резерв
; L88
LOAD      P01322	// OUT: Резерв
OR        M0008A	// FORCE IN: Резерв
OUT       M0003A	// Резерв
; L90
LOAD      P01323	// OUT: Резерв
OR        M0008B	// FORCE IN: Резерв
OUT       M0003B	// Резерв
; L92
LOAD      P01324	// OUT: Резерв
OR        M0008C	// FORCE IN: Резерв
OUT       M0003C	// Резерв
; L94
LOAD      P01325	// OUT: Резерв
OR        M0008D	// FORCE IN: Резерв
OUT       M0003D	// Резерв
; L96
LOAD      P01326	// OUT: Резерв
OR        M0008E	// FORCE IN: Резерв
OUT       M0003E	// Резерв
; L98
LOAD      P01327	// OUT: Резерв
OR        M0008F	// FORCE IN: Резерв
OUT       M0003F	// Резерв

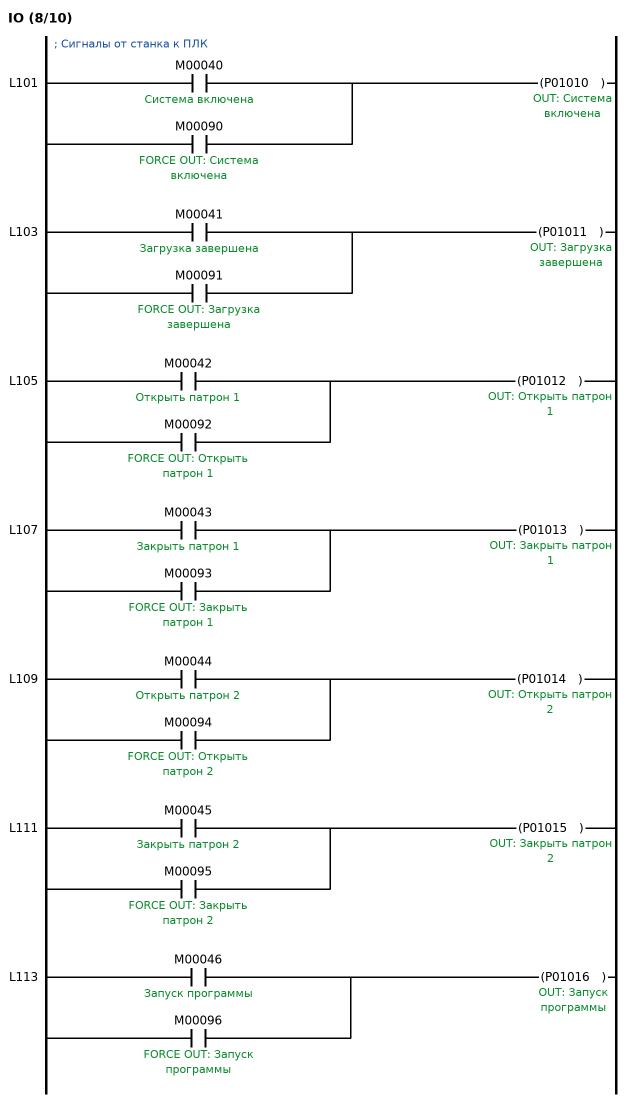
// Сигналы от станка к ПЛК
; L101
LOAD      M00040	// Система включена
OR        M00090	// FORCE OUT: Система включена
OUT       P01010	// OUT: Система включена
; L103
LOAD      M00041	// Загрузка завершена
OR        M00091	// FORCE OUT: Загрузка завершена
OUT       P01011	// OUT: Загрузка завершена
; L105
LOAD      M00042	// Открыть патрон 1
OR        M00092	// FORCE OUT: Открыть патрон 1
OUT       P01012	// OUT: Открыть патрон 1
; L107
LOAD      M00043	// Закрыть патрон 1
OR        M00093	// FORCE OUT: Закрыть патрон 1
OUT       P01013	// OUT: Закрыть патрон 1
; L109
LOAD      M00044	// Открыть патрон 2
OR        M00094	// FORCE OUT: Открыть патрон 2
OUT       P01014	// OUT: Открыть патрон 2
; L111
LOAD      M00045	// Закрыть патрон 2
OR        M00095	// FORCE OUT: Закрыть патрон 2
OUT       P01015	// OUT: Закрыть патрон 2
; L113
LOAD      M00046	// Запуск программы
OR        M00096	// FORCE OUT: Запуск программы
OUT       P01016	// OUT: Запуск программы

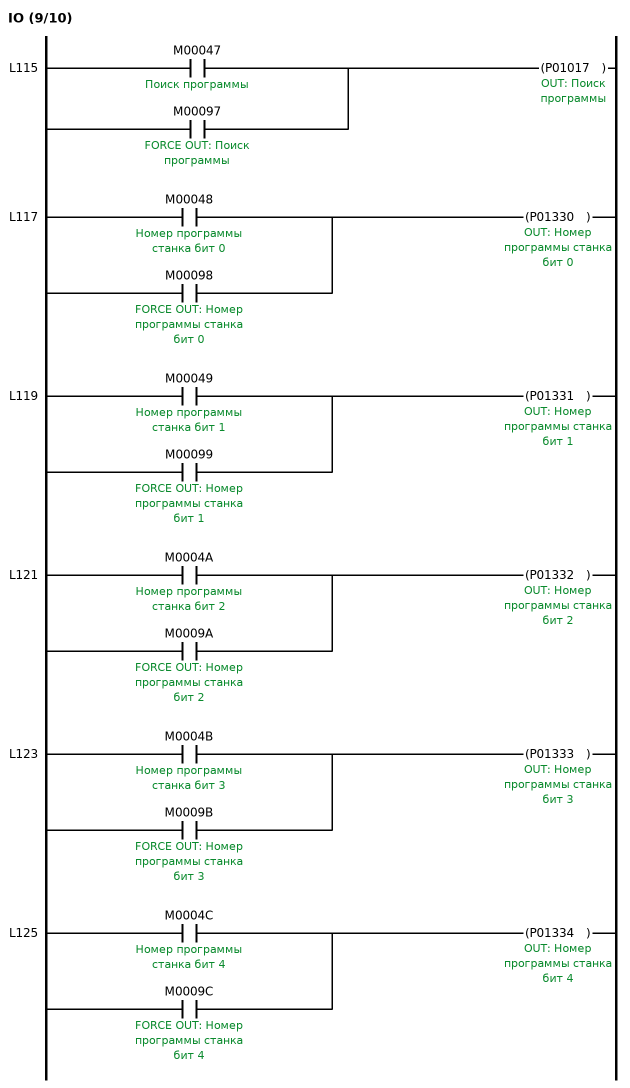
; L115
LOAD      M00047	// Поиск программы
OR        M00097	// FORCE OUT: Поиск программы
OUT       P01017	// OUT: Поиск программы
; L117
LOAD      M00048	// Номер программы станка бит 0
OR        M00098	// FORCE OUT: Номер программы станка бит 0
OUT       P01330	// OUT: Номер программы станка бит 0
; L119
LOAD      M00049	// Номер программы станка бит 1
OR        M00099	// FORCE OUT: Номер программы станка бит 1
OUT       P01331	// OUT: Номер программы станка бит 1
; L121
LOAD      M0004A	// Номер программы станка бит 2
OR        M0009A	// FORCE OUT: Номер программы станка бит 2
OUT       P01332	// OUT: Номер программы станка бит 2
; L123
LOAD      M0004B	// Номер программы станка бит 3
OR        M0009B	// FORCE OUT: Номер программы станка бит 3
OUT       P01333	// OUT: Номер программы станка бит 3
; L125
LOAD      M0004C	// Номер программы станка бит 4
OR        M0009C	// FORCE OUT: Номер программы станка бит 4
OUT       P01334	// OUT: Номер программы станка бит 4

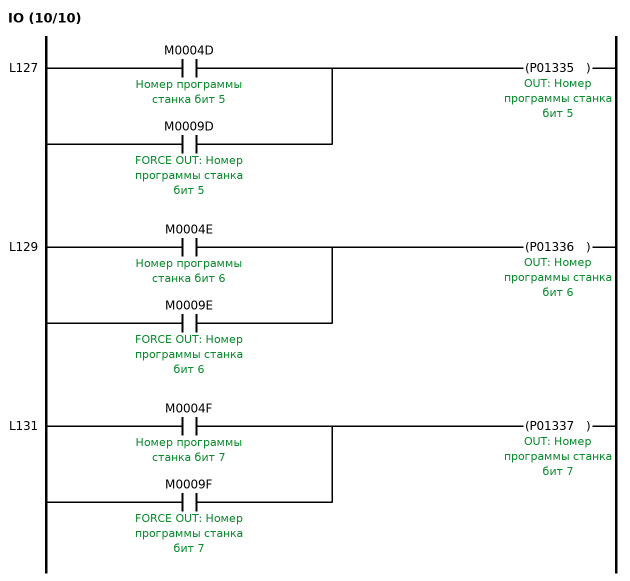
; L127
LOAD      M0004D	// Номер программы станка бит 5
OR        M0009D	// FORCE OUT: Номер программы станка бит 5
OUT       P01335	// OUT: Номер программы станка бит 5
; L129
LOAD      M0004E	// Номер программы станка бит 6
OR        M0009E	// FORCE OUT: Номер программы станка бит 6
OUT       P01336	// OUT: Номер программы станка бит 6
; L131
LOAD      M0004F	// Номер программы станка бит 7
OR        M0009F	// FORCE OUT: Номер программы станка бит 7
OUT       P01337	// OUT: Номер программы станка бит 7

PROGRAM Error (task: Scan Program)

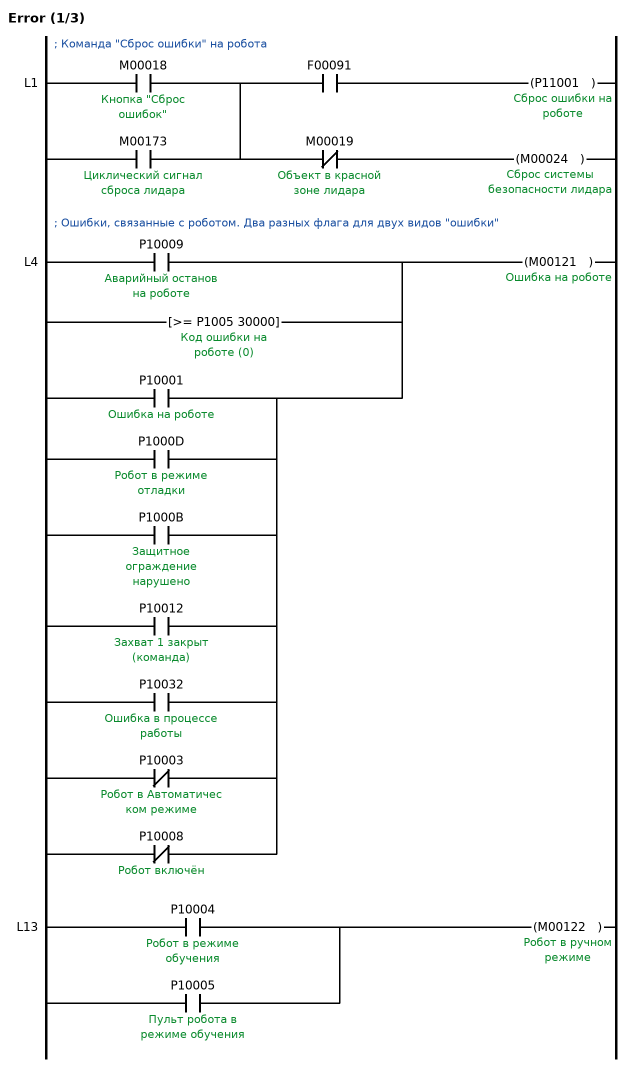
// Команда "Сброс ошибки" на робота
; L1
LOAD      M00018	// Кнопка "Сброс ошибок"
OR        M00173	// Циклический сигнал сброса лидара
MPUSH
AND       F00091
OUT       P11001	// Сброс ошибки на роботе
MPOP
AND NOT   M00019	//  Объект в красной зоне лидара
OUT       M00024	// Сброс системы безопасности лидара
// Ошибки, связанные с роботом. Два разных флага для двух видов "ошибки"
; L4
LOAD      P10009	// Аварийный останов на роботе
OR>=      P1005 30000	// Код ошибки на роботе (0)
OR        P10001	// Ошибка на роботе
OR        P1000D	// Робот в режиме отладки
OR        P1000B	// Защитное ограждение нарушено
OR        P10012	// Захват 1 закрыт (команда)
OR        P10032	// Ошибка в процессе работы
OR NOT    P10003	// Робот в Автоматическом режиме
OR NOT    P10008	// Робот включён
OUT       M00121	// Ошибка на роботе
; L13
LOAD      P10004	// Робот в режиме обучения
OR        P10005	// Пульт робота в режиме обучения
OUT       M00122	// Робот в ручном режиме

